FUNCTION TryConvert_LWORD_TO_LINT : BOOL
VAR_INPUT
	in : LWORD;
	out : REFERENCE TO LINT;
END_VAR

IF in > DatatypeLimits.MAX_VALUE_OF_LWORD_WHICH_CAN_BE_HELD_IN_A_LINT THEN
	RETURN;
END_IF

out := LWORD_TO_LINT(in);
TryConvert_LWORD_TO_LINT := TRUE;

END_FUNCTION

(* stored: Version 1.1.0.1, ProductVersion 3.1.4024.12
   POU TryConvert_LWORD_TO_LINT: Id {4e7fe53b-ac55-436b-a89f-019271eada18}, SpecialFunc None *)
